// TIA Portal V20 export
VAR_GLOBAL   // PLC tag table "Default tag table"
   GateIN_Safety1_1 AT %I5050.0 : Bool;
   GateOUT_Safety2_1 AT %I5050.1 : Bool;
   Door_Safety3_1 AT %I5050.2 : Bool;
   Szafa_15_Safety4_1 AT %I5050.3 : Bool;
   GateIN_Safety1_2 AT %I5050.4 : Bool;
   GateOUT_Safety2_2 AT %I5050.5 : Bool;
   Door_Safety3_2 AT %I5050.6 : Bool;
   Szafa15_Safety4_2 AT %I5050.7 : Bool;
   Clock_Byte AT %MB0 : Byte;
   Clock_10Hz AT %M0.0 : Bool;
   Clock_5Hz AT %M0.1 : Bool;
   "Clock_2.5Hz" AT %M0.2 : Bool;
   Clock_2Hz AT %M0.3 : Bool;
   "Clock_1.25Hz" AT %M0.4 : Bool;
   Clock_1Hz AT %M0.5 : Bool;
   "Clock_0.625Hz" AT %M0.6 : Bool;
   "Clock_0.5Hz" AT %M0.7 : Bool;
   Tag_1 AT %ID5200 : DInt;
END_VAR
